(* PLC project Practical Work One, Rexroth ctrlX PLC Engineering ctrlX PLC 1.16.1, author Cedric Lenoir *)
(* stored: creationDateTime 2024-02-29T13:48:24.1388527, version 0.0, modificationDateTime 2024-02-29T13:41:03.804153, organization HEVS *)
(* First Test for Practical Work One *)

TYPE UA_DigitalInput_32 : STRUCT
  Input_0_0 : BOOL;
  Input_0_1 : BOOL;
  Input_0_2 : BOOL;
  Input_0_3 : BOOL;
  Input_0_4 : BOOL;
  Input_0_5 : BOOL;
  Input_0_6 : BOOL;
  Input_0_7 : BOOL;
  Input_1_0 : BOOL;
  Input_1_1 : BOOL;
  Input_1_2 : BOOL;
  Input_1_3 : BOOL;
  Input_1_4 : BOOL;
  Input_1_5 : BOOL;
  Input_1_6 : BOOL;
  Input_1_7 : BOOL;
  Input_2_0 : BOOL;
  Input_2_1 : BOOL;
  Input_2_2 : BOOL;
  Input_2_3 : BOOL;
  Input_2_4 : BOOL;
  Input_2_5 : BOOL;
  Input_2_6 : BOOL;
  Input_2_7 : BOOL;
  Input_3_0 : BOOL;
  Input_3_1 : BOOL;
  Input_3_2 : BOOL;
  Input_3_3 : BOOL;
  Input_3_4 : BOOL;
  Input_3_5 : BOOL;
  Input_3_6 : BOOL;
  Input_3_7 : BOOL;
END_STRUCT;
END_TYPE

TYPE UA_DigitalOutput_32 : STRUCT
  Output_0_0 : BOOL;
  Output_0_1 : BOOL;
  Output_0_2 : BOOL;
  Output_0_3 : BOOL;
  Output_0_4 : BOOL;
  Output_0_5 : BOOL;
  Output_0_6 : BOOL;
  Output_0_7 : BOOL;
  Output_1_0 : BOOL;
  Output_1_1 : BOOL;
  Output_1_2 : BOOL;
  Output_1_3 : BOOL;
  Output_1_4 : BOOL;
  Output_1_5 : BOOL;
  Output_1_6 : BOOL;
  Output_1_7 : BOOL;
  Output_2_0 : BOOL;
  Output_2_1 : BOOL;
  Output_2_2 : BOOL;
  Output_2_3 : BOOL;
  Output_2_4 : BOOL;
  Output_2_5 : BOOL;
  Output_2_6 : BOOL;
  Output_2_7 : BOOL;
  Output_3_0 : BOOL;
  Output_3_1 : BOOL;
  Output_3_2 : BOOL;
  Output_3_3 : BOOL;
  Output_3_4 : BOOL;
  Output_3_5 : BOOL;
  Output_3_6 : BOOL;
  Output_3_7 : BOOL;
END_STRUCT;
END_TYPE

TYPE UA_ButtonAndSignal : STRUCT
  In_Estop : BOOL;
  In_Reset : BOOL;
  In_Start : BOOL;
  In_Stop : BOOL;
  Out_Idle : BOOL;
  Out_Execute : BOOL;
  Out_Stopped : BOOL;
END_STRUCT;
END_TYPE

TYPE UA_O300_DL : STRUCT
  Value : WORD;
  BCD1 : BOOL;
  Q : BOOL;
  A : BOOL;
END_STRUCT;
END_TYPE

TYPE UA_O300_ZL : STRUCT
  BCD1 : BOOL;
  Q : BOOL;
  A : BOOL;
END_STRUCT;
END_TYPE

TYPE UA_U300_D50 : STRUCT
  Value : DWORD;
  Scale : SINT;
  SSC1 : BOOL;
  SSC2 : BOOL;
  Q : BOOL;
  A : BOOL;
  SSC4 : BOOL;
END_STRUCT;
END_TYPE

TYPE UA_U300_P50 : STRUCT
  Value : DWORD;
  Scale : SINT;
  SSC1 : BOOL;
  SSC2 : BOOL;
  Q : BOOL;
  A : BOOL;
  SSC4 : BOOL;
END_STRUCT;
END_TYPE

TYPE UA_Schunk_mms : STRUCT
  Value : WORD;
END_STRUCT;
END_TYPE

TYPE UA_Balluf_bcm0002 : STRUCT
  Data_1 : REAL;
  Data_2 : REAL;
  Data_3 : REAL;
  Temperature : REAL;
  Status : DWORD;
END_STRUCT;
END_TYPE

TYPE UA_Festo : STRUCT
  SetOut : BOOL;
END_STRUCT;
END_TYPE

TYPE UA_AnalogIn : STRUCT
  IW_04 : WORD;
  IW_06 : WORD;
  IW_08 : WORD;
  IW_10 : WORD;
  IW_12 : WORD;
  IW_14 : WORD;
  IW_16 : WORD;
  IW_18 : WORD;
END_STRUCT;
END_TYPE

TYPE UA_AnalogOut : STRUCT
  QW_04 : WORD;
  QW_06 : WORD;
  QW_08 : WORD;
  QW_10 : WORD;
END_STRUCT;
END_TYPE

TYPE UA_AboxInterface : STRUCT
  uaButtonAndSignal : UA_ButtonAndSignal;
  uaAnalogIn : UA_AnalogIn;
  uaAnalogOut : UA_AnalogOut;
  uaDigitalIn : UA_DigitalInput_32;
  uaDigitalOut : UA_DigitalOutput_32;
  uaO300_DL_Optic : UA_O300_DL;
  uaO300_ZL_Optic : UA_O300_ZL;
  uaU300_D50_Sound : UA_U300_D50;
  uaU300_P50_Sound : UA_U300_P50;
  uaSchunk : UA_Schunk_mms;
  uaSchunkGripper : UA_Festo;
  uaAccelerometer : UA_Balluf_bcm0002;
END_STRUCT;
END_TYPE

(* www.hevs.ch Institut Systemes Industriels Project: Projet No: PW Move Absolute Author: Cedric Lenoir Date: 2023 October 16 Summary: List of commands for MoveAbsolute *)
TYPE ST_PlcOpenFbs : STRUCT
  bEnableRemote : BOOL;  (* If TRUE, the FB are driven manually from the HMI *)
  bEnableReadStatus : BOOL;
  bEnableReadPosition : BOOL;
  bEnableReadVelocity : BOOL;
  bMoveAbs : BOOL;
  bStop : BOOL;
  bPowerOn : BOOL;
  bReset : BOOL;
  strGetAxisStatus : STRING;  (* From arAxisStatus_gb[1].Data.PLCopenState; Exist in Data Layer too, s=motion/axs/Axis_X/state/opstate/plcopen *)
END_STRUCT;
END_TYPE

(* www.hevs.ch Institut Systemes Industriels Project: Projet No: PW Move Absolute Author: Cedric Lenoir Date: 2023 October 16 Summary: List of dynamic parameters for Move Absolute *)
TYPE ST_SetMotionParam : STRUCT
  rPosition_mm : LREAL;
  rVeloctiy_mm_s : LREAL;
  rAcceleration_mm_s2 : LREAL;
  rDeceleration_mm_s2 : LREAL;
  rJerk_mm_s3 : LREAL;
END_STRUCT;
END_TYPE

(* www.hevs.ch Institut Systemes Industriels Project: Projet No: PW Move Absolute Author: Cedric Lenoir Date: 2023 October 16 Summary: State Machine Info *)
TYPE ST_StateMachineInfo : STRUCT
  diState : DINT;
  eState : EN_MoveAbsStates;
  bIdle : BOOL;
  bActive : BOOL;
  bError : BOOL;
  strState : STRING;
END_STRUCT;
END_TYPE

(* www.hevs.ch Institut Systemes Industriels Project: Projet No: PW Move Absolute Author: Cedric Lenoir Date: 2024 February 29 Summary: Template of a program using PLCopen for motion *)
PROGRAM PLC_PRG
  VAR
    uliCount : ULINT;
    bInitDone : BOOL;
    stPlcOpenFbs : ST_PlcOpenFbs;  (* List of Structures *)
    stSetMotionParam : ST_SetMotionParam := (rVeloctiy_mm_s := 100, rAcceleration_mm_s2 := 1000, rDeceleration_mm_s2 := 1000, rJerk_mm_s3 := 1000);
    stStateMachineInfo : ST_StateMachineInfo;
    mcReadActualPosition : MC_ReadActualPosition;  (* List of Function Blocks *)
    mcReadActualVelocity : MC_ReadActualVelocity;
    mcReadStatus : MC_ReadStatus;
    mcPower : MC_Power;  (* On va essayer de changer la position de référence (Hors tension) mcHome : MC_Home; not possible, check for a set reference mise sous tension standard *)
    mcMoveAbsolute : MC_MoveAbsolute;  (* Simplement trois mouvemements différents *)
    mcStop : MC_Stop := (Deceleration := 1);  (* On va essayer d'arreter l'axe suffisament rapidement pour le STO *)
    mcReset : MC_Reset;
  END_VAR

                    (*
    Some inits independant of the Main State Machine
*)
IF NOT bInitDone THEN
	bInitDone := TRUE;
    stPlcOpenFbs.bEnableReadStatus := TRUE;
    stPlcOpenFbs.bEnableReadPosition := TRUE;
    stPlcOpenFbs.bEnableReadVelocity := TRUE;
END_IF

(*
    Remote conditions
*)
IF stPlcOpenFbs.bEnableRemote THEN
    IF mcMoveAbsolute.Done THEN
        stPlcOpenFbs.bMoveAbs := FALSE;
    END_IF
    IF mcStop.Done THEN
        stPlcOpenFbs.bStop := FALSE;
        stPlcOpenFbs.bMoveAbs := FALSE;
    END_IF
END_IF

(*
    Main State Machine.
*)
CASE stStateMachineInfo.eState OF
    EN_MoveAbsStates.eIdle :
        stStateMachineInfo.strState := 'Idle';
        ;
    EN_MoveAbsStates.eIsPowerOff :
        stStateMachineInfo.strState := 'Is Power Off';
        ;
    EN_MoveAbsStates.eWaitPowerOn :
        stStateMachineInfo.strState := 'Wait for Power On';
        ;
    EN_MoveAbsStates.eIsPowerOn :
        stStateMachineInfo.strState := 'Is Power On';
        ;
    EN_MoveAbsStates.eInitMotion :
        stStateMachineInfo.strState := 'Motion Init active';
        ;
    EN_MoveAbsStates.eInitMotionDone :
        stStateMachineInfo.strState := 'Motion Init done';
        ;
    EN_MoveAbsStates.eStopping :
        stStateMachineInfo.strState := 'Stopping active';
        ;
    EN_MoveAbsStates.eMoveDown :
        stStateMachineInfo.strState := 'Move Down active';
        ;
    EN_MoveAbsStates.eMoveDownDone :
        stStateMachineInfo.strState := 'Move Down done';
        ;
    EN_MoveAbsStates.eCloseGripper :
        stStateMachineInfo.strState := 'Close Gripper active';
        ;
    EN_MoveAbsStates.eGripperClosed :
        stStateMachineInfo.strState := 'Close Gripper done';
        ;
    EN_MoveAbsStates.eErrorStop :
        stStateMachineInfo.strState := 'Is in Error Stop';
        ;
END_CASE
(*
    Get state machine in a DINT format
*)
stStateMachineInfo.diState := stStateMachineInfo.eState;
(*
    Error state depends only of the state machine in combinational logic.
    That is, some Booleans are defined solely based on a combination of states.
*) 
stStateMachineInfo.bIdle := stStateMachineInfo.eState = EN_MoveAbsStates.eIdle;
stStateMachineInfo.bError := stStateMachineInfo.eState = EN_MoveAbsStates.eErrorStop;
stStateMachineInfo.bActive := NOT (stStateMachineInfo.eState = EN_MoveAbsStates.eIdle) AND
                              NOT (stStateMachineInfo.eState = EN_MoveAbsStates.eErrorStop);

(*
    Call all Function Blocks at the end of the program
    This is a good practice.
*)
mcReadStatus(Axis := GVL_AxisDefines.X_Axis,
             Enable := stPlcOpenFbs.bEnableReadStatus);

mcReadActualPosition(Axis := GVL_AxisDefines.X_Axis,
                     Enable := stPlcOpenFbs.bEnableReadPosition);
                                         
mcReadActualVelocity(Axis := GVL_AxisDefines.X_Axis,
                     Enable := stPlcOpenFbs.bEnableReadVelocity);

mcPower(Axis := GVL_AxisDefines.X_Axis,
        Enable := stPlcOpenFbs.bPowerOn);

mcMoveAbsolute(Axis := GVL_AxisDefines.X_Axis,
               Position := stSetMotionParam.rPosition_mm,
               Velocity := stSetMotionParam.rVeloctiy_mm_s,
               Acceleration := stSetMotionParam.rAcceleration_mm_s2,
               Deceleration := stSetMotionParam.rDeceleration_mm_s2,
               Jerk := stSetMotionParam.rJerk_mm_s3,
               Execute := stPlcOpenFbs.bMoveAbs);               

// A noter que un stop sans décélération conduit à une erreur !
mcStop(Axis := GVL_AxisDefines.X_Axis,
       Execute := stPlcOpenFbs.bStop);

mcReset(Axis := GVL_AxisDefines.X_Axis,
        Execute := stPlcOpenFbs.bReset);
                   
                  
END_PROGRAM

PROGRAM PRG_MapBox
  VAR
    UA_ReadCounterFromStation : DINT;  (* Write from Siemens to ctrX Core Used to check if read is running *)
    UA_ButtonAndSignal_In_Estop : BOOL;
    UA_ButtonAndSignal_In_Reset : BOOL;
    UA_ButtonAndSignal_In_Start : BOOL;
    UA_ButtonAndSignal_In_Stop : BOOL;
    UA_Balluf_bcm0002_Data_1 : REAL;
    UA_Balluf_bcm0002_Data_2 : REAL;
    UA_Balluf_bcm0002_Data_3 : REAL;
    UA_Balluf_bcm0002_Temperature : REAL;
    UA_Balluf_bcm0002_Status : DWORD;
    UA_Festo_SetOut : BOOL;
    UA_O300_DL_Value : WORD;
    UA_O300_DL_BCD1 : BOOL;
    UA_O300_DL_Q : BOOL;
    UA_O300_DL_A : BOOL;
    UA_O300_ZL_BCD1 : BOOL;
    UA_O300_ZL_Q : BOOL;
    UA_O300_ZL_A : BOOL;
    UA_U300_D50_Value : DWORD;
    UA_U300_D50_Scale : SINT;
    UA_U300_D50_SSC1 : BOOL;
    UA_U300_D50_SSC2 : BOOL;
    UA_U300_D50_Q : BOOL;
    UA_U300_D50_A : BOOL;
    UA_U300_D50_SSC4 : BOOL;
    UA_U300_P50_Value : DWORD;
    UA_U300_P50_Scale : SINT;
    UA_U300_P50_SSC1 : BOOL;
    UA_U300_P50_SSC2 : BOOL;
    UA_U300_P50_Q : BOOL;
    UA_U300_P50_A : BOOL;
    UA_U300_P50_SSC4 : BOOL;
    UA_DigitalInput_32_Input_0_0 : BOOL;
    UA_DigitalInput_32_Input_0_1 : BOOL;
    UA_DigitalInput_32_Input_0_2 : BOOL;
    UA_DigitalInput_32_Input_0_3 : BOOL;
    UA_DigitalInput_32_Input_0_4 : BOOL;
    UA_DigitalInput_32_Input_0_5 : BOOL;
    UA_DigitalInput_32_Input_0_6 : BOOL;
    UA_DigitalInput_32_Input_0_7 : BOOL;
    UA_DigitalInput_32_Input_1_0 : BOOL;
    UA_DigitalInput_32_Input_1_1 : BOOL;
    UA_DigitalInput_32_Input_1_2 : BOOL;
    UA_DigitalInput_32_Input_1_3 : BOOL;
    UA_DigitalInput_32_Input_1_4 : BOOL;
    UA_DigitalInput_32_Input_1_5 : BOOL;
    UA_DigitalInput_32_Input_1_6 : BOOL;
    UA_DigitalInput_32_Input_1_7 : BOOL;
    UA_DigitalInput_32_Input_2_0 : BOOL;
    UA_DigitalInput_32_Input_2_1 : BOOL;
    UA_DigitalInput_32_Input_2_2 : BOOL;
    UA_DigitalInput_32_Input_2_3 : BOOL;
    UA_DigitalInput_32_Input_2_4 : BOOL;
    UA_DigitalInput_32_Input_2_5 : BOOL;
    UA_DigitalInput_32_Input_2_6 : BOOL;
    UA_DigitalInput_32_Input_2_7 : BOOL;
    UA_DigitalInput_32_Input_3_0 : BOOL;
    UA_DigitalInput_32_Input_3_1 : BOOL;
    UA_DigitalInput_32_Input_3_2 : BOOL;
    UA_DigitalInput_32_Input_3_3 : BOOL;
    UA_DigitalInput_32_Input_3_4 : BOOL;
    UA_DigitalInput_32_Input_3_5 : BOOL;
    UA_DigitalInput_32_Input_3_6 : BOOL;
    UA_DigitalInput_32_Input_3_7 : BOOL;
    UA_WriteCounterToStation : DINT;  (* Siemens Read from ctrX Core Used to check if write is running *)
    UA_ButtonAndSignal_Out_Idle : BOOL;
    UA_ButtonAndSignal_Out_Execute : BOOL;
    UA_ButtonAndSignal_Out_Stopped : BOOL;
    UA_Schunk_mms_Value : WORD;
    UA_DigitalOutput_32_Output_0_0 : BOOL;
    UA_DigitalOutput_32_Output_0_1 : BOOL;
    UA_DigitalOutput_32_Output_0_2 : BOOL;
    UA_DigitalOutput_32_Output_0_3 : BOOL;
    UA_DigitalOutput_32_Output_0_4 : BOOL;
    UA_DigitalOutput_32_Output_0_5 : BOOL;
    UA_DigitalOutput_32_Output_0_6 : BOOL;
    UA_DigitalOutput_32_Output_0_7 : BOOL;
    UA_DigitalOutput_32_Output_1_0 : BOOL;
    UA_DigitalOutput_32_Output_1_1 : BOOL;
    UA_DigitalOutput_32_Output_1_2 : BOOL;
    UA_DigitalOutput_32_Output_1_3 : BOOL;
    UA_DigitalOutput_32_Output_1_4 : BOOL;
    UA_DigitalOutput_32_Output_1_5 : BOOL;
    UA_DigitalOutput_32_Output_1_6 : BOOL;
    UA_DigitalOutput_32_Output_1_7 : BOOL;
    UA_DigitalOutput_32_Output_2_0 : BOOL;
    UA_DigitalOutput_32_Output_2_1 : BOOL;
    UA_DigitalOutput_32_Output_2_2 : BOOL;
    UA_DigitalOutput_32_Output_2_3 : BOOL;
    UA_DigitalOutput_32_Output_2_4 : BOOL;
    UA_DigitalOutput_32_Output_2_5 : BOOL;
    UA_DigitalOutput_32_Output_2_6 : BOOL;
    UA_DigitalOutput_32_Output_2_7 : BOOL;
    UA_DigitalOutput_32_Output_3_0 : BOOL;
    UA_DigitalOutput_32_Output_3_1 : BOOL;
    UA_DigitalOutput_32_Output_3_2 : BOOL;
    UA_DigitalOutput_32_Output_3_3 : BOOL;
    UA_DigitalOutput_32_Output_3_4 : BOOL;
    UA_DigitalOutput_32_Output_3_5 : BOOL;
    UA_DigitalOutput_32_Output_3_6 : BOOL;
    UA_DigitalOutput_32_Output_3_7 : BOOL;
  END_VAR

                        (*
        Values from Profinet Station
    *)
    
    // Get Value from Profinet Station with UA Client Write
	GVL_Abox.uaAboxInterface.uaButtonAndSignal.In_Estop     := UA_ButtonAndSignal_In_Estop;
	GVL_Abox.uaAboxInterface.uaButtonAndSignal.In_Reset     := UA_ButtonAndSignal_In_Reset;
	GVL_Abox.uaAboxInterface.uaButtonAndSignal.In_Start     := UA_ButtonAndSignal_In_Start;
	GVL_Abox.uaAboxInterface.uaButtonAndSignal.In_Stop      := UA_ButtonAndSignal_In_Stop;
    // Values from Balluff accelerometer
    GVL_Abox.uaAboxInterface.uaAccelerometer.Data_1         := UA_Balluf_bcm0002_Data_1;
    GVL_Abox.uaAboxInterface.uaAccelerometer.Data_2         := UA_Balluf_bcm0002_Data_1;
    GVL_Abox.uaAboxInterface.uaAccelerometer.Data_3         := UA_Balluf_bcm0002_Data_1;
    GVL_Abox.uaAboxInterface.uaAccelerometer.Status         := UA_Balluf_bcm0002_Status;
    GVL_Abox.uaAboxInterface.uaAccelerometer.Temperature    := UA_Balluf_bcm0002_Temperature;

    // Values from Baumer O300 DL
    GVL_Abox.uaAboxInterface.uaO300_DL_Optic.Value          := UA_O300_DL_Value;                
    GVL_Abox.uaAboxInterface.uaO300_DL_Optic.A              := UA_O300_DL_A;                
    GVL_Abox.uaAboxInterface.uaO300_DL_Optic.Q              := UA_O300_DL_Q;                
    GVL_Abox.uaAboxInterface.uaO300_DL_Optic.BCD1           := UA_O300_DL_BCD1;                

    // Values from Baumer O300 ZL                
    GVL_Abox.uaAboxInterface.uaO300_ZL_Optic.A              := UA_O300_ZL_A;                
    GVL_Abox.uaAboxInterface.uaO300_ZL_Optic.Q              := UA_O300_ZL_Q;                
    GVL_Abox.uaAboxInterface.uaO300_ZL_Optic.BCD1           := UA_O300_ZL_BCD1;                

    // Values from Baumer U300 D50
    GVL_Abox.uaAboxInterface.uaU300_D50_Sound.Value         := UA_U300_D50_Value;  
    GVL_Abox.uaAboxInterface.uaU300_D50_Sound.A             := UA_U300_D50_A;  
    GVL_Abox.uaAboxInterface.uaU300_D50_Sound.Q             := UA_U300_D50_Q;  
    GVL_Abox.uaAboxInterface.uaU300_D50_Sound.Scale         := UA_U300_D50_Scale;  
    GVL_Abox.uaAboxInterface.uaU300_D50_Sound.SSC1          := UA_U300_D50_SSC1;  
    GVL_Abox.uaAboxInterface.uaU300_D50_Sound.SSC2          := UA_U300_D50_SSC2;  
    GVL_Abox.uaAboxInterface.uaU300_D50_Sound.SSC4          := UA_U300_D50_SSC4;  
    
    // Values from Baumer U300 P50
    GVL_Abox.uaAboxInterface.uaU300_P50_Sound.Value         := UA_U300_P50_Value;  
    GVL_Abox.uaAboxInterface.uaU300_P50_Sound.A             := UA_U300_P50_A;  
    GVL_Abox.uaAboxInterface.uaU300_P50_Sound.Q             := UA_U300_P50_Q;  
    GVL_Abox.uaAboxInterface.uaU300_P50_Sound.Scale         := UA_U300_P50_Scale;  
    GVL_Abox.uaAboxInterface.uaU300_P50_Sound.SSC1          := UA_U300_P50_SSC1;  
    GVL_Abox.uaAboxInterface.uaU300_P50_Sound.SSC2          := UA_U300_P50_SSC2;  
    GVL_Abox.uaAboxInterface.uaU300_P50_Sound.SSC4          := UA_U300_P50_SSC4;  
    
    // Values from Gripper sensor
    GVL_Abox.uaAboxInterface.uaSchunk.Value                 := UA_Schunk_mms_Value;  
    
    // Get 32 Digital Input
    GVL_Abox.uaAboxInterface.uaDigitalIn.Input_0_0          := UA_DigitalInput_32_Input_0_0;
    GVL_Abox.uaAboxInterface.uaDigitalIn.Input_0_1          := UA_DigitalInput_32_Input_0_1;
    GVL_Abox.uaAboxInterface.uaDigitalIn.Input_0_2          := UA_DigitalInput_32_Input_0_2;
    GVL_Abox.uaAboxInterface.uaDigitalIn.Input_0_3          := UA_DigitalInput_32_Input_0_3;
    GVL_Abox.uaAboxInterface.uaDigitalIn.Input_0_4          := UA_DigitalInput_32_Input_0_4;
    GVL_Abox.uaAboxInterface.uaDigitalIn.Input_0_5          := UA_DigitalInput_32_Input_0_5;
    GVL_Abox.uaAboxInterface.uaDigitalIn.Input_0_6          := UA_DigitalInput_32_Input_0_6;
    GVL_Abox.uaAboxInterface.uaDigitalIn.Input_0_7          := UA_DigitalInput_32_Input_0_7;
    GVL_Abox.uaAboxInterface.uaDigitalIn.Input_1_0          := UA_DigitalInput_32_Input_1_0;
    GVL_Abox.uaAboxInterface.uaDigitalIn.Input_1_1          := UA_DigitalInput_32_Input_1_1;
    GVL_Abox.uaAboxInterface.uaDigitalIn.Input_1_2          := UA_DigitalInput_32_Input_1_2;
    GVL_Abox.uaAboxInterface.uaDigitalIn.Input_1_3          := UA_DigitalInput_32_Input_1_3;
    GVL_Abox.uaAboxInterface.uaDigitalIn.Input_1_4          := UA_DigitalInput_32_Input_1_4;
    GVL_Abox.uaAboxInterface.uaDigitalIn.Input_1_5          := UA_DigitalInput_32_Input_1_5;
    GVL_Abox.uaAboxInterface.uaDigitalIn.Input_1_6          := UA_DigitalInput_32_Input_1_6;
    GVL_Abox.uaAboxInterface.uaDigitalIn.Input_1_7          := UA_DigitalInput_32_Input_1_7;
    GVL_Abox.uaAboxInterface.uaDigitalIn.Input_2_0          := UA_DigitalInput_32_Input_2_0;
    GVL_Abox.uaAboxInterface.uaDigitalIn.Input_2_1          := UA_DigitalInput_32_Input_2_1;
    GVL_Abox.uaAboxInterface.uaDigitalIn.Input_2_2          := UA_DigitalInput_32_Input_2_2;
    GVL_Abox.uaAboxInterface.uaDigitalIn.Input_2_3          := UA_DigitalInput_32_Input_2_3;
    GVL_Abox.uaAboxInterface.uaDigitalIn.Input_2_4          := UA_DigitalInput_32_Input_2_4;
    GVL_Abox.uaAboxInterface.uaDigitalIn.Input_2_5          := UA_DigitalInput_32_Input_2_5;
    GVL_Abox.uaAboxInterface.uaDigitalIn.Input_2_6          := UA_DigitalInput_32_Input_2_6;
    GVL_Abox.uaAboxInterface.uaDigitalIn.Input_2_7          := UA_DigitalInput_32_Input_2_7;
    GVL_Abox.uaAboxInterface.uaDigitalIn.Input_3_0          := UA_DigitalInput_32_Input_3_0;
    GVL_Abox.uaAboxInterface.uaDigitalIn.Input_3_1          := UA_DigitalInput_32_Input_3_1;
    GVL_Abox.uaAboxInterface.uaDigitalIn.Input_3_2          := UA_DigitalInput_32_Input_3_2;
    GVL_Abox.uaAboxInterface.uaDigitalIn.Input_3_3          := UA_DigitalInput_32_Input_3_3;
    GVL_Abox.uaAboxInterface.uaDigitalIn.Input_3_4          := UA_DigitalInput_32_Input_3_4;
    GVL_Abox.uaAboxInterface.uaDigitalIn.Input_3_5          := UA_DigitalInput_32_Input_3_5;
    GVL_Abox.uaAboxInterface.uaDigitalIn.Input_3_6          := UA_DigitalInput_32_Input_3_6;
    GVL_Abox.uaAboxInterface.uaDigitalIn.Input_3_7          := UA_DigitalInput_32_Input_3_7;
    
    (*
        Values to Profinet Station
    *)
	UA_WriteCounterToStation := UA_WriteCounterToStation + 1;

    // Set Visual Signals
	UA_ButtonAndSignal_Out_Execute 	:= GVL_Abox.uaAboxInterface.uaButtonAndSignal.Out_Execute;
	UA_ButtonAndSignal_Out_Idle 	:= GVL_Abox.uaAboxInterface.uaButtonAndSignal.Out_Idle;
	UA_ButtonAndSignal_Out_Stopped	:= GVL_Abox.uaAboxInterface.uaButtonAndSignal.Out_Stopped;
    
    // Set Gripper value
    UA_Festo_SetOut                 := GVL_Abox.uaAboxInterface.uaSchunkGripper.SetOut;
    
    // Set 32 digital outputs
    UA_DigitalOutput_32_Output_0_0  := GVL_Abox.uaAboxInterface.uaDigitalOut.Output_0_0;
    UA_DigitalOutput_32_Output_0_1  := GVL_Abox.uaAboxInterface.uaDigitalOut.Output_0_1;
    UA_DigitalOutput_32_Output_0_2  := GVL_Abox.uaAboxInterface.uaDigitalOut.Output_0_2;
    UA_DigitalOutput_32_Output_0_3  := GVL_Abox.uaAboxInterface.uaDigitalOut.Output_0_3;
    UA_DigitalOutput_32_Output_0_4  := GVL_Abox.uaAboxInterface.uaDigitalOut.Output_0_4;
    UA_DigitalOutput_32_Output_0_5  := GVL_Abox.uaAboxInterface.uaDigitalOut.Output_0_5;
    UA_DigitalOutput_32_Output_0_6  := GVL_Abox.uaAboxInterface.uaDigitalOut.Output_0_6;
    UA_DigitalOutput_32_Output_0_7  := GVL_Abox.uaAboxInterface.uaDigitalOut.Output_0_7;
    UA_DigitalOutput_32_Output_1_0  := GVL_Abox.uaAboxInterface.uaDigitalOut.Output_1_0;
    UA_DigitalOutput_32_Output_1_1  := GVL_Abox.uaAboxInterface.uaDigitalOut.Output_1_1;
    UA_DigitalOutput_32_Output_1_2  := GVL_Abox.uaAboxInterface.uaDigitalOut.Output_1_2;
    UA_DigitalOutput_32_Output_1_3  := GVL_Abox.uaAboxInterface.uaDigitalOut.Output_1_3;
    UA_DigitalOutput_32_Output_1_4  := GVL_Abox.uaAboxInterface.uaDigitalOut.Output_1_4;
    UA_DigitalOutput_32_Output_1_5  := GVL_Abox.uaAboxInterface.uaDigitalOut.Output_1_5;
    UA_DigitalOutput_32_Output_1_6  := GVL_Abox.uaAboxInterface.uaDigitalOut.Output_1_6;
    UA_DigitalOutput_32_Output_1_7  := GVL_Abox.uaAboxInterface.uaDigitalOut.Output_1_7;
    UA_DigitalOutput_32_Output_2_0  := GVL_Abox.uaAboxInterface.uaDigitalOut.Output_2_0;
    UA_DigitalOutput_32_Output_2_1  := GVL_Abox.uaAboxInterface.uaDigitalOut.Output_2_1;
    UA_DigitalOutput_32_Output_2_2  := GVL_Abox.uaAboxInterface.uaDigitalOut.Output_2_2;
    UA_DigitalOutput_32_Output_2_3  := GVL_Abox.uaAboxInterface.uaDigitalOut.Output_2_3;
    UA_DigitalOutput_32_Output_2_4  := GVL_Abox.uaAboxInterface.uaDigitalOut.Output_2_4;
    UA_DigitalOutput_32_Output_2_5  := GVL_Abox.uaAboxInterface.uaDigitalOut.Output_2_5;
    UA_DigitalOutput_32_Output_2_6  := GVL_Abox.uaAboxInterface.uaDigitalOut.Output_2_6;
    UA_DigitalOutput_32_Output_2_7  := GVL_Abox.uaAboxInterface.uaDigitalOut.Output_2_7;
    UA_DigitalOutput_32_Output_3_0  := GVL_Abox.uaAboxInterface.uaDigitalOut.Output_3_0;
    UA_DigitalOutput_32_Output_3_1  := GVL_Abox.uaAboxInterface.uaDigitalOut.Output_3_1;
    UA_DigitalOutput_32_Output_3_2  := GVL_Abox.uaAboxInterface.uaDigitalOut.Output_3_2;
    UA_DigitalOutput_32_Output_3_3  := GVL_Abox.uaAboxInterface.uaDigitalOut.Output_3_3;
    UA_DigitalOutput_32_Output_3_4  := GVL_Abox.uaAboxInterface.uaDigitalOut.Output_3_4;
    UA_DigitalOutput_32_Output_3_5  := GVL_Abox.uaAboxInterface.uaDigitalOut.Output_3_5;
    UA_DigitalOutput_32_Output_3_6  := GVL_Abox.uaAboxInterface.uaDigitalOut.Output_3_6;
    UA_DigitalOutput_32_Output_3_7  := GVL_Abox.uaAboxInterface.uaDigitalOut.Output_3_7;
    
PRG_CHECK_IO();
                  
END_PROGRAM

PROGRAM PRG_CHECK_IO
  VAR
    testButton_1 : BOOL;
    testButton_2 : BOOL;
    testButton_3 : BOOL;
    clignote : TON;
    changeMeSlow : BOOL;
    clignoteSlow : TON;
    changeMe : BOOL;
    NotResetTest : BOOL := TRUE;
  END_VAR

                    testButton_1 := GVL_Abox.uaAboxInterface.uaButtonAndSignal.In_Reset;
testButton_2 := GVL_Abox.uaAboxInterface.uaButtonAndSignal.In_Start;
testButton_3 := GVL_Abox.uaAboxInterface.uaButtonAndSignal.In_Stop;

IF GVL_Abox.uaAboxInterface.uaButtonAndSignal.In_Reset AND
   NotResetTest										   THEN
	NotResetTest := FALSE;
	
    GVL_Abox.uaAboxInterface.uaSchunkGripper.SetOut := FALSE;
    
    GVL_Abox.uaAboxInterface.uaButtonAndSignal.Out_Execute := FALSE;	
    GVL_Abox.uaAboxInterface.uaButtonAndSignal.Out_Idle := FALSE;	
    GVL_Abox.uaAboxInterface.uaButtonAndSignal.Out_Stopped := FALSE;	

    GVL_Abox.uaAboxInterface.uaDigitalOut.Output_0_0 := FALSE;
    GVL_Abox.uaAboxInterface.uaDigitalOut.Output_0_1 := FALSE;
    GVL_Abox.uaAboxInterface.uaDigitalOut.Output_0_2 := FALSE;
    GVL_Abox.uaAboxInterface.uaDigitalOut.Output_0_3 := FALSE;
    GVL_Abox.uaAboxInterface.uaDigitalOut.Output_0_4 := FALSE;
    GVL_Abox.uaAboxInterface.uaDigitalOut.Output_0_5 := FALSE;
    GVL_Abox.uaAboxInterface.uaDigitalOut.Output_0_6 := FALSE;
    GVL_Abox.uaAboxInterface.uaDigitalOut.Output_0_7 := FALSE;
    
    GVL_Abox.uaAboxInterface.uaDigitalOut.Output_1_0 := FALSE;
    GVL_Abox.uaAboxInterface.uaDigitalOut.Output_1_1 := FALSE;
    GVL_Abox.uaAboxInterface.uaDigitalOut.Output_1_2 := FALSE;
    GVL_Abox.uaAboxInterface.uaDigitalOut.Output_1_3 := FALSE;
    GVL_Abox.uaAboxInterface.uaDigitalOut.Output_1_4 := FALSE;
    GVL_Abox.uaAboxInterface.uaDigitalOut.Output_1_5 := FALSE;
    GVL_Abox.uaAboxInterface.uaDigitalOut.Output_1_6 := FALSE;
    GVL_Abox.uaAboxInterface.uaDigitalOut.Output_1_7 := FALSE;
    
    GVL_Abox.uaAboxInterface.uaDigitalOut.Output_2_0 := FALSE;
    GVL_Abox.uaAboxInterface.uaDigitalOut.Output_2_1 := FALSE;
    GVL_Abox.uaAboxInterface.uaDigitalOut.Output_2_2 := FALSE;
    GVL_Abox.uaAboxInterface.uaDigitalOut.Output_2_3 := FALSE;
    GVL_Abox.uaAboxInterface.uaDigitalOut.Output_2_4 := FALSE;
    GVL_Abox.uaAboxInterface.uaDigitalOut.Output_2_5 := FALSE;
    GVL_Abox.uaAboxInterface.uaDigitalOut.Output_2_6 := FALSE;
    GVL_Abox.uaAboxInterface.uaDigitalOut.Output_2_7 := FALSE;

    GVL_Abox.uaAboxInterface.uaDigitalOut.Output_3_0 := FALSE;
    GVL_Abox.uaAboxInterface.uaDigitalOut.Output_3_1 := FALSE;
    GVL_Abox.uaAboxInterface.uaDigitalOut.Output_3_2 := FALSE;
    GVL_Abox.uaAboxInterface.uaDigitalOut.Output_3_3 := FALSE;
    GVL_Abox.uaAboxInterface.uaDigitalOut.Output_3_4 := FALSE;
    GVL_Abox.uaAboxInterface.uaDigitalOut.Output_3_5 := FALSE;
    GVL_Abox.uaAboxInterface.uaDigitalOut.Output_3_6 := FALSE;
    GVL_Abox.uaAboxInterface.uaDigitalOut.Output_3_7 := FALSE;	
END_IF

IF GVL_Abox.uaAboxInterface.uaButtonAndSignal.In_Reset AND
   GVL_Abox.uaAboxInterface.uaButtonAndSignal.In_Start AND
   GVL_Abox.uaAboxInterface.uaButtonAndSignal.In_Stop  THEN
	NotResetTest := TRUE;
END_IF


IF NotResetTest THEN 
	
	// Quick Blink
	clignote(IN := changeMe,
			 PT := T#500MS);
			 
	IF clignote.Q THEN
		changeMe := FALSE;
	ELSE
		changeMe := TRUE;
	END_IF

	// Slow Blink
	clignoteSlow(IN := changeMeSlow,
			 	 PT := T#2500MS);
			 
	IF clignoteSlow.Q THEN
		changeMeSlow := FALSE;
	ELSE
		changeMeSlow := TRUE;
	END_IF
	
	IF (NOT GVL_Abox.uaAboxInterface.uaSchunkGripper.SetOut) AND clignoteSlow.Q THEN
		GVL_Abox.uaAboxInterface.uaSchunkGripper.SetOut := TRUE;
	ELSIF GVL_Abox.uaAboxInterface.uaSchunkGripper.SetOut AND clignoteSlow.Q THEN
		GVL_Abox.uaAboxInterface.uaSchunkGripper.SetOut := FALSE;
	END_IF
	
	IF (NOT GVL_Abox.uaAboxInterface.uaDigitalOut.Output_0_0) AND clignote.Q THEN
		GVL_Abox.uaAboxInterface.uaButtonAndSignal.Out_Execute := TRUE;	
		GVL_Abox.uaAboxInterface.uaButtonAndSignal.Out_Idle := TRUE;	
		GVL_Abox.uaAboxInterface.uaButtonAndSignal.Out_Stopped := TRUE;	
	
		GVL_Abox.uaAboxInterface.uaDigitalOut.Output_0_0 := TRUE;
		GVL_Abox.uaAboxInterface.uaDigitalOut.Output_0_1 := TRUE;
		GVL_Abox.uaAboxInterface.uaDigitalOut.Output_0_2 := TRUE;
		GVL_Abox.uaAboxInterface.uaDigitalOut.Output_0_3 := TRUE;
		GVL_Abox.uaAboxInterface.uaDigitalOut.Output_0_4 := TRUE;
		GVL_Abox.uaAboxInterface.uaDigitalOut.Output_0_5 := TRUE;
		GVL_Abox.uaAboxInterface.uaDigitalOut.Output_0_6 := TRUE;
		GVL_Abox.uaAboxInterface.uaDigitalOut.Output_0_7 := TRUE;
		
		GVL_Abox.uaAboxInterface.uaDigitalOut.Output_1_0 := TRUE;
		GVL_Abox.uaAboxInterface.uaDigitalOut.Output_1_1 := TRUE;
		GVL_Abox.uaAboxInterface.uaDigitalOut.Output_1_2 := TRUE;
		GVL_Abox.uaAboxInterface.uaDigitalOut.Output_1_3 := TRUE;
		GVL_Abox.uaAboxInterface.uaDigitalOut.Output_1_4 := TRUE;
		GVL_Abox.uaAboxInterface.uaDigitalOut.Output_1_5 := TRUE;
		GVL_Abox.uaAboxInterface.uaDigitalOut.Output_1_6 := TRUE;
		GVL_Abox.uaAboxInterface.uaDigitalOut.Output_1_7 := TRUE;
		
		GVL_Abox.uaAboxInterface.uaDigitalOut.Output_2_0 := TRUE;
		GVL_Abox.uaAboxInterface.uaDigitalOut.Output_2_1 := TRUE;
		GVL_Abox.uaAboxInterface.uaDigitalOut.Output_2_2 := TRUE;
		GVL_Abox.uaAboxInterface.uaDigitalOut.Output_2_3 := TRUE;
		GVL_Abox.uaAboxInterface.uaDigitalOut.Output_2_4 := TRUE;
		GVL_Abox.uaAboxInterface.uaDigitalOut.Output_2_5 := TRUE;
		GVL_Abox.uaAboxInterface.uaDigitalOut.Output_2_6 := TRUE;
		GVL_Abox.uaAboxInterface.uaDigitalOut.Output_2_7 := TRUE;

		GVL_Abox.uaAboxInterface.uaDigitalOut.Output_3_0 := TRUE;
		GVL_Abox.uaAboxInterface.uaDigitalOut.Output_3_1 := TRUE;
		GVL_Abox.uaAboxInterface.uaDigitalOut.Output_3_2 := TRUE;
		GVL_Abox.uaAboxInterface.uaDigitalOut.Output_3_3 := TRUE;
		GVL_Abox.uaAboxInterface.uaDigitalOut.Output_3_4 := TRUE;
		GVL_Abox.uaAboxInterface.uaDigitalOut.Output_3_5 := TRUE;
		GVL_Abox.uaAboxInterface.uaDigitalOut.Output_3_6 := TRUE;
		GVL_Abox.uaAboxInterface.uaDigitalOut.Output_3_7 := TRUE;
	ELSIF GVL_Abox.uaAboxInterface.uaDigitalOut.Output_0_0 AND clignote.Q THEN
		GVL_Abox.uaAboxInterface.uaButtonAndSignal.Out_Execute := FALSE;	
		GVL_Abox.uaAboxInterface.uaButtonAndSignal.Out_Idle := FALSE;	
		GVL_Abox.uaAboxInterface.uaButtonAndSignal.Out_Stopped := FALSE;	

		GVL_Abox.uaAboxInterface.uaDigitalOut.Output_0_0 := FALSE;
		GVL_Abox.uaAboxInterface.uaDigitalOut.Output_0_1 := FALSE;
		GVL_Abox.uaAboxInterface.uaDigitalOut.Output_0_2 := FALSE;
		GVL_Abox.uaAboxInterface.uaDigitalOut.Output_0_3 := FALSE;
		GVL_Abox.uaAboxInterface.uaDigitalOut.Output_0_4 := FALSE;
		GVL_Abox.uaAboxInterface.uaDigitalOut.Output_0_5 := FALSE;
		GVL_Abox.uaAboxInterface.uaDigitalOut.Output_0_6 := FALSE;
		GVL_Abox.uaAboxInterface.uaDigitalOut.Output_0_7 := FALSE;
		
		GVL_Abox.uaAboxInterface.uaDigitalOut.Output_1_0 := FALSE;
		GVL_Abox.uaAboxInterface.uaDigitalOut.Output_1_1 := FALSE;
		GVL_Abox.uaAboxInterface.uaDigitalOut.Output_1_2 := FALSE;
		GVL_Abox.uaAboxInterface.uaDigitalOut.Output_1_3 := FALSE;
		GVL_Abox.uaAboxInterface.uaDigitalOut.Output_1_4 := FALSE;
		GVL_Abox.uaAboxInterface.uaDigitalOut.Output_1_5 := FALSE;
		GVL_Abox.uaAboxInterface.uaDigitalOut.Output_1_6 := FALSE;
		GVL_Abox.uaAboxInterface.uaDigitalOut.Output_1_7 := FALSE;
		
		GVL_Abox.uaAboxInterface.uaDigitalOut.Output_2_0 := FALSE;
		GVL_Abox.uaAboxInterface.uaDigitalOut.Output_2_1 := FALSE;
		GVL_Abox.uaAboxInterface.uaDigitalOut.Output_2_2 := FALSE;
		GVL_Abox.uaAboxInterface.uaDigitalOut.Output_2_3 := FALSE;
		GVL_Abox.uaAboxInterface.uaDigitalOut.Output_2_4 := FALSE;
		GVL_Abox.uaAboxInterface.uaDigitalOut.Output_2_5 := FALSE;
		GVL_Abox.uaAboxInterface.uaDigitalOut.Output_2_6 := FALSE;
		GVL_Abox.uaAboxInterface.uaDigitalOut.Output_2_7 := FALSE;

		GVL_Abox.uaAboxInterface.uaDigitalOut.Output_3_0 := FALSE;
		GVL_Abox.uaAboxInterface.uaDigitalOut.Output_3_1 := FALSE;
		GVL_Abox.uaAboxInterface.uaDigitalOut.Output_3_2 := FALSE;
		GVL_Abox.uaAboxInterface.uaDigitalOut.Output_3_3 := FALSE;
		GVL_Abox.uaAboxInterface.uaDigitalOut.Output_3_4 := FALSE;
		GVL_Abox.uaAboxInterface.uaDigitalOut.Output_3_5 := FALSE;
		GVL_Abox.uaAboxInterface.uaDigitalOut.Output_3_6 := FALSE;
		GVL_Abox.uaAboxInterface.uaDigitalOut.Output_3_7 := FALSE;
	END_IF;
END_IF
                  
END_PROGRAM

CONFIGURATION PracticalWork_01
  RESOURCE BaseInterfaceUa ON PLC
    {attribute 'qualified_only'}
    VAR_GLOBAL  (* GVL_Abox *)
      uaAboxInterface : UA_AboxInterface;
    END_VAR
    {attribute 'qualified_only'}
    VAR_GLOBAL  (* GVL_Unit *)
      myConveyor : ST_Conveyor;
      myHmi : ST_HmiConveyor;
    END_VAR
    {attribute 'qualified_only'}
    VAR_GLOBAL  (* GVL_AxisDefines *)
      X_Axis : MB_AXISIF_REF := (AxisName := 'Axis_1', AxisNo := 1);
    END_VAR
    TASK MainTask(INTERVAL := T#10ms, PRIORITY := 30);
    PROGRAM PLC_PRG WITH MainTask : PLC_PRG;
    PROGRAM PRG_MapBox WITH MainTask : PRG_MapBox;
  END_RESOURCE
END_CONFIGURATION

CONFIGURATION Realtime_Data
END_CONFIGURATION
